TYPE LAxisCtrl_typeGeneralSettings :
STRUCT

	stopOnError			:BOOL;
	resetWithRestart			:BOOL;
	abortWaitingSyncCmd		:BOOL;

END_STRUCT
END_TYPE

(* stored: Version 1.1.0.1
   DUT LAxisCtrl_typeGeneralSettings: Id {b47046e5-6b99-498b-b166-53e3252fbdf7} *)
